// Gets the upper bound index of the array of specified type.
FUNCTION F_GetUIntArrayUpperBound : T_Position // The upper bound index of the specified array.
VAR_IN_OUT
	arArray : ARRAY[*] OF UINT; // The array to query.
END_VAR

F_GetUIntArrayUpperBound := UPPER_BOUND(arArray, 1);

END_FUNCTION

(* stored: Version 1.1.0.1
   POU F_GetUIntArrayUpperBound: Id {29caff58-0eb2-0ad9-3358-90ecab558fce}, SpecialFunc None *)
